// Mitsubishi GX Works2 project: 030923 ex fblock soma sub   PLC: Q03UDV

// task Task_01 (event TRUE, interval 0, priority 31): POU_01
// task Tarefa1 (event TRUE, interval 0, priority 31): 

PROGRAM POU_01
VAR
  fSubtração_1 : INT;
END_VAR
(* structured ladder/FBD written out as ST: instructions are called as NAME(EN, inputs, outputs); _pN, _eN, _tN stand for wires *)
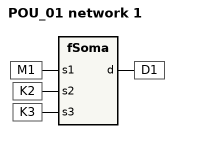
(* network 1 *)
D1 := fSoma(M1, K2, K3);
END_PROGRAM

FUNCTION fSoma
VAR_INPUT
  i_xHabilitar : BOOL;
  i_iElemento1 : INT;
  i_iElemento2 : INT;
END_VAR
(* structured ladder/FBD written out as ST: instructions are called as NAME(EN, inputs, outputs); _pN, _eN, _tN stand for wires *)
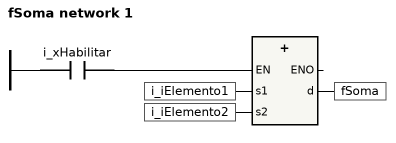
(* network 1 *)
+(i_xHabilitar, i_iElemento1, i_iElemento2, fSoma);
END_FUNCTION

PROGRAM ST_Example
VAR
  XEnable : BOOL;
END_VAR
VAR CONSTANT
  i_iElemento1 : INT := 1;
  i_iElemento2 : INT := 2;
END_VAR
VAR
  iDR : ARRAY [0..1] OF INT;
  iDR1 : ARRAY [0..1] OF DINT;
  xEnableOperacao : BOOL;
  XEnableOperacao2 : BOOL;
  xEnableOperacao3 : BOOL;
  iValorValidar : BOOL;
  iContador : BOOL;
END_VAR
iDR[0]:= fSoma( XEnable, i_iElemento1 , i_iElemento2);
iDR[1]:= fSubstraction( XEnable, i_iElemento1,i_iElemento2);
iDR1[0]:=fMultiplication( XEnable , i_iElement1, i_iElement2 );

(*******************************************************)
IF  xEnableOperacao AND NOT xEnableOperacao3  THEN
	 iDR[1]:= fSubstraction( XEnable, i_iElemento1,i_iElemento2);
ELSE IF XEnableOperacao2
	 iDR[0]:= fSoma( XEnable, i_iElemento1 , i_iElemento2);
END_IF;

(*******************************************************)
CASE  iValorValidar  OF
	 0:
		  iDR[0]:= fSoma( XEnable, i_iElemento1 , i_iElemento2);
	 1,2:
		  iDR[0]:= fSoma( XEnable, i_iElemento1 , i_iElemento2);
	 3..5:
		  iDR[0]:= fSoma( XEnable, i_iElemento1 , i_iElemento2);
	ELSE
		  iDR[0]:= fSoma( XEnable, i_iElemento1 , i_iElemento2);

END_CASE;

(********************************************)
FOR  iContador := 0  TO  10  BY  1  DO
	  iDR[0]:= fSoma( XEnable, i_iElemento1 , i_iElemento2) ;
END_FOR;
END_PROGRAM

FUNCTION fSubstraction
VAR_INPUT
  i_Elemento1 : INT;
  i_Elemento2 : INT;
  i_Enable : BOOL;
END_VAR
(* structured ladder/FBD written out as ST: instructions are called as NAME(EN, inputs, outputs); _pN, _eN, _tN stand for wires *)
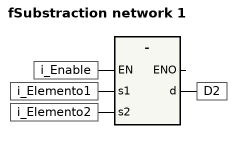
(* network 1 *)
-(i_Enable, i_Elemento1, i_Elemento2, D2);
END_FUNCTION

FUNCTION fMultiplication
VAR_INPUT
  i_Enable : BOOL;
  i_Element1 : INT;
  i_Element2 : INT;
END_VAR
(* structured ladder/FBD written out as ST: instructions are called as NAME(EN, inputs, outputs); _pN, _eN, _tN stand for wires *)
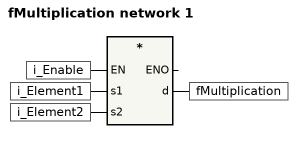
(* network 1 *)
*(i_Enable, i_Element1, i_Element2, fMultiplication);
END_FUNCTION
